FUNCTION_BLOCK BasicAdapter (* Basic FB with empty ECC *)
  (* Standard: 61499-2 *)
  (* Version 1.0, 2023-03-07, AK115394 *)
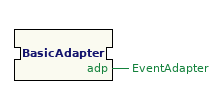
  PLUGS
    adp : EventAdapter;
  END_PLUGS
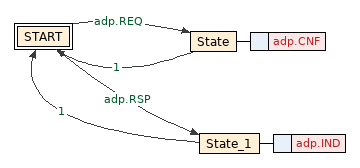
  EC_STATES
    START; (* Initial State *)
    State : -> adp.CNF;
    State_1 : -> adp.IND;
  END_STATES
  EC_TRANSITIONS
    START TO State := adp.REQ;
    State TO START := 1;
    START TO State_1 := adp.RSP;
    State_1 TO START := 1;
  END_TRANSITIONS
END_FUNCTION_BLOCK
